(* PLC project Hydraulic Simulator Functions library, Porcheson Hydraulic Simulator 0.0 *)
(* stored: creationDateTime 2023-02-10T00:00:00, modificationDateTime 2026-02-10T00:00:00 *)

FUNCTION_BLOCK HYD_CreateSimAxis
  VAR_INPUT
    AXISTYPE : USINT;
    MAXVEL : REAL;
    MAXACC : REAL;
    MAXDEC : REAL;
  END_VAR
  VAR_OUTPUT
    AXISID : SINT;
    DONE : BOOL;
  END_VAR

						{{ extern void __mcl_cmd_createSimAxis(HYD_CREATESIMAXIS *data__);	__mcl_cmd_createSimAxis(data__);	 }}	
					
END_FUNCTION_BLOCK

FUNCTION_BLOCK HYD_MoveSimAxis
  VAR_INPUT
    ENABLE : BOOL;
    AXISID : SINT;
    CMD_RPM : REAL;
    DIRECTION : SINT;
  END_VAR
  VAR_OUTPUT
    BUSY : BOOL;
  END_VAR

						{{ extern void __mcl_cmd_moveSimAxis(HYD_MOVESIMAXIS *data__);	__mcl_cmd_moveSimAxis(data__);	 }}	
					
END_FUNCTION_BLOCK

FUNCTION_BLOCK HYD_ReadSimAxis
  VAR_INPUT
    ENABLE : BOOL;
    AXISID : SINT;
  END_VAR
  VAR_OUTPUT
    ACTIVE : BOOL;
    POS_MM : REAL;
    VEL_MM_S : REAL;
    PRESSURE_BAR : REAL;
    BUSY : BOOL;
  END_VAR

						{{ extern void __mcl_cmd_readSimAxis(HYD_READSIMAXIS *data__);	__mcl_cmd_readSimAxis(data__);	 }}	
					
END_FUNCTION_BLOCK
